(* PLC project Adressering.ecp, WAGO e!COCKPIT e!COCKPIT *)
(* stored: creationDateTime 2021-01-18T14:20:23.2110188, modificationDateTime 2021-01-18T11:51:27.6823754 *)

TYPE typVAV : STRUCT
  xReady : BOOL;  (* Status adr. *)
  xEnable : BOOL;  (* Enable MP blokk *)
  xAddress : BOOL;  (* Adresserer VAV *)
  xFailed : BOOL;  (* Tilbakemelding adressering (True = SerieNr inn og ut ikke stemmer) *)
  sSetStatus : STRING;  (* Status tilbakemelding naar adresseringen er i SET step *)
  sGetStatus : STRING;  (* Status tilbakemelding naar adresseringen er i GET step *)
  iSerialNr : typSerialNo;  (* Serie NR *)
  bPort : BYTE;  (* VAV Port *)
  bAddress : BYTE;  (* VAV Address *)
  rAirVolume_SP : REAL;  (* Settpunkt 0-100% *)
  rOutPosition : REAL;  (* Vinkel *)
  rOutAirVolume_perc : REAL;  (* Luftmengde i prosent *)
  rOutAirVolume_m3h : REAL;  (* Luftmengde i m3h *)
  wSensorValue : WORD;
  rVmin : REAL;
  rVmax : REAL;  (* Max vinkel *)
  xControlRangeIncreased : BOOL;
  xMecanicalOverload : BOOL;
  xActuatorHunting : BOOL;
  xSensorError : BOOL;
  xManualOpen : BOOL;
  xManualClose : BOOL;
  vMin : REAL;  (* Min luftmengde SP / 0-100 *)
  vNorm : REAL;  (* Settpunkt ved bevegelse / 0-100 *)
  vMax : REAL;  (* Maks luftmengde SP / 0-100 *)
  vSize : REAL;  (* Max kubikk *)
  vSetpoint_m3h : REAL;  (* SP% *)
  xdontoptimize : BOOL;  (* Fjerner VAV fra Optimizer *)
END_STRUCT;
END_TYPE

{attribute 'qualified_only'}
VAR_GLOBAL  (* STLV80_360 *)
  STLV80_A_360_6D201_SQ401 : typVAV := (xEnable := TRUE, vMin := 700, vNorm := 1400, vMax := 1400, vSize := 1750, bPort := 1, bAddress := 1, iSerialNr := (wYearAndWeek := 02045, wDayAndNumber := 50010, bTypeID := 158, bTestStation := 140));  (* / *)
  STLV80_A_360_6D301_SQ501 : typVAV := (xEnable := TRUE, vMin := 3200, vNorm := 3200, vMax := 3200, vSize := 5655, bPort := 1, bAddress := 2, iSerialNr := (wYearAndWeek := 02040, wDayAndNumber := 40202, bTypeID := 158, bTestStation := 153));  (* / *)
  STLV80_A_360_6A201_SQ401 : typVAV := (xEnable := TRUE, vMin := 2025, vNorm := 4050, vMax := 4050, vSize := 5655, bPort := 1, bAddress := 3, iSerialNr := (wYearAndWeek := 02040, wDayAndNumber := 40197, bTypeID := 158, bTestStation := 140));  (* / *)
  STLV80_A_360_6A201_SQ501 : typVAV := (xEnable := TRUE, vMin := 2700, vNorm := 2700, vMax := 2700, vSize := 5655, bPort := 1, bAddress := 4, iSerialNr := (wYearAndWeek := 02040, wDayAndNumber := 40201, bTypeID := 158, bTestStation := 159));  (* / *)
  STLV80_A_360_6C206_SQ501 : typVAV := (xEnable := TRUE, vMin := 300, vNorm := 300, vMax := 300, vSize := 700, bPort := 1, bAddress := 5, iSerialNr := (wYearAndWeek := 02105, wDayAndNumber := 10009, bTypeID := 158, bTestStation := 142));  (* / *)
  STLV80_A_360_6C206_SQ401 : typVAV := (xEnable := TRUE, vMin := 375, vNorm := 750, vMax := 750, vSize := 1750, bPort := 1, bAddress := 6, iSerialNr := (wYearAndWeek := 02045, wDayAndNumber := 50010, bTypeID := 158, bTestStation := 153));  (* / *)
  STLV80_A_360_7C201_SQ401 : typVAV := (xEnable := TRUE, vMin := 200, vNorm := 200, vMax := 200, vSize := 434, bPort := 1, bAddress := 7, iSerialNr := (wYearAndWeek := 02032, wDayAndNumber := 40145, bTypeID := 158, bTestStation := 158));  (* / *)
  STLV80_A_360_7C201_SQ501 : typVAV := (xEnable := TRUE, vMin := 400, vNorm := 400, vMax := 400, vSize := 700, bPort := 1, bAddress := 8, iSerialNr := (wYearAndWeek := 02042, wDayAndNumber := 10210, bTypeID := 158, bTestStation := 153));  (* / *)
  STLV80_A_360_6G201_SQ401 : typVAV := (xEnable := TRUE, vMin := 700, vNorm := 1400, vMax := 1400, vSize := 3619, bPort := 2, bAddress := 1, iSerialNr := (wYearAndWeek := 02042, wDayAndNumber := 10209, bTypeID := 158, bTestStation := 153));  (* / *)
  STLV80_A_360_6M201_SQ503 : typVAV := (xEnable := TRUE, vMin := 850, vNorm := 850, vMax := 850, vSize := 1060, bPort := 2, bAddress := 2, iSerialNr := (wYearAndWeek := 02005, wDayAndNumber := 20125, bTypeID := 158, bTestStation := 140));  (* / *)
  STLV80_A_360_6M201_SQ403 : typVAV := (xEnable := TRUE, vMin := 1225, vNorm := 2450, vMax := 2450, vSize := 5344, bPort := 2, bAddress := 3, iSerialNr := (wYearAndWeek := 02045, wDayAndNumber := 20003, bTypeID := 158, bTestStation := 140));  (* / *)
  STLV80_A_360_6M201_SQ402 : typVAV := (xEnable := TRUE, vMin := 700, vNorm := 1400, vMax := 1400, vSize := 4524, bPort := 2, bAddress := 4, iSerialNr := (wYearAndWeek := 02042, wDayAndNumber := 10207, bTypeID := 158, bTestStation := 153));  (* / *)
  STLV80_A_360_6M201_SQ502 : typVAV := (xEnable := TRUE, vMin := 3850, vNorm := 3850, vMax := 3850, vSize := 5655, bPort := 2, bAddress := 5, iSerialNr := (wYearAndWeek := 02040, wDayAndNumber := 40196, bTypeID := 158, bTestStation := 140));  (* / *)
  STLV80_A_360_6M201_SQ501 : typVAV := (xEnable := TRUE, vMin := 2600, vNorm := 2600, vMax := 2600, vSize := 5655, bPort := 2, bAddress := 6, iSerialNr := (wYearAndWeek := 02044, wDayAndNumber := 00121, bTypeID := 158, bTestStation := 164));  (* / *)
  STLV80_A_360_6M201_SQ401 : typVAV := (xEnable := TRUE, vMin := 900, vNorm := 1800, vMax := 1800, vSize := 5344, bPort := 2, bAddress := 7, iSerialNr := (wYearAndWeek := 02045, wDayAndNumber := 20006, bTypeID := 158, bTestStation := 140));  (* / *)
  STLV80_A_360_7O201_SQ401 : typVAV := (xEnable := TRUE, vMin := 200, vNorm := 200, vMax := 200, vSize := 700, bPort := 3, bAddress := 1, iSerialNr := (wYearAndWeek := 02032, wDayAndNumber := 40155, bTypeID := 158, bTestStation := 129));  (* / *)
  STLV80_A_360_7O201_SQ501 : typVAV := (xEnable := TRUE, vMin := 400, vNorm := 400, vMax := 400, vSize := 700, bPort := 3, bAddress := 2, iSerialNr := (wYearAndWeek := 02049, wDayAndNumber := 40093, bTypeID := 158, bTestStation := 142));  (* / *)
END_VAR

FUNCTION_BLOCK fbAutAd
  VAR_INPUT
    iSerialNr : typSerialNo;
    bPort : BYTE;
    bAddress : BYTE;
    xReset : BOOL;
    xNext : BOOL;
  END_VAR
  VAR_OUTPUT
    i : INT := 0;
    xFailed : BOOL;
    sSetStatus : STRING;
    sGetStatus : STRING;
  END_VAR
  VAR
    xLearn : BOOL;
    xRetry : BOOL;
    VAV_Addressing : fbMpBusAddressing;
  END_VAR

	//Resetter forgje VAVs verdier
	IF xReset THEN
		i:= 0;
		xRetry:= FALSE;
		xFailed:= FALSE;
		sSetStatus:= '';
		sGetStatus:= '';

//Begynner paa neste VAV
	ELSIF i<1 AND xNext THEN
		VAV_Addressing
		(
			bPortMpBus:= bPort,
			bAddress:= bAddress,
			typINSerialNo:= iSerialNr,
			xLearn:= xLearn
		);
		i:= 1;

//Skriver rett port og adresse til VAV naar blokken er klar
	ELSIF VAV_Addressing.xReady AND i=1 THEN
		VAV_Addressing
		(
			xSet:= TRUE,
			xLearn:= xLearn
		);
		i:= 2;

//Spoer etter serie nr som hoerer til port og adresse
	ELSIF VAV_Addressing.xReady AND i=2 THEN
		sSetStatus:= VAV_Addressing.sStatus;
		VAV_Addressing
		(
			xGetSerialNO:= TRUE,
			xLearn:= xLearn
		);
		i:= 3;

//Sjekker om serie nr. som tilhoerer port og adressen stemmer
	ELSIF VAV_Addressing.xReady AND i=3 THEN
		sGetStatus:= VAV_Addressing.sStatus;
		//Sjekker om serie nr stemmer
		IF xRetry AND VAV_Addressing.typOUTSerialNo.wYearAndWeek <> iSerialNr.wYearAndWeek OR VAV_Addressing.typOUTSerialNo.wDayAndNumber <> iSerialNr.wDayAndNumber OR VAV_Addressing.typOUTSerialNo.bTypeID <> iSerialNr.bTypeID OR VAV_Addressing.typOUTSerialNo.bTestStation <> iSerialNr.bTestStation THEN
			xRetry:= FALSE;
			xFailed:= TRUE;
			i:=4;
		ELSIF VAV_Addressing.typOUTSerialNo.wYearAndWeek <> iSerialNr.wYearAndWeek OR VAV_Addressing.typOUTSerialNo.wDayAndNumber <> iSerialNr.wDayAndNumber OR VAV_Addressing.typOUTSerialNo.bTypeID <> iSerialNr.bTypeID OR VAV_Addressing.typOUTSerialNo.bTestStation <> iSerialNr.bTestStation THEN
			xRetry:= TRUE;
			i:=1;
		ELSE
			i:=4;
		END_IF

//Resetter xSet og xGet, og Setter Port, adresse og serie nr. og henter status
	ELSE
		VAV_Addressing
		(
			bPortMpBus:= bPort,
			bAddress:= bAddress,
			typINSerialNo:= iSerialNr,
			xLearn:= xLearn,
			xSet:= FALSE,
			xGetSerialNO:= FALSE,
			xLearn:= xLearn
		);
	END_IF
				
END_FUNCTION_BLOCK

PROGRAM PRG_VAV_Adressering
  VAR
    xReset : BOOL;
    xRun : BOOL;
    xInit : BOOL := TRUE;
    Auto : fbAutAd;
    iLinje : INT;  (* Linje som skal adresseres *)
    iVAV : INT := 1;  (* VAV(adr.) som adresseres *)
  END_VAR

					IF xReset THEN
	Auto(xReset:= TRUE);
	xInit:= TRUE;
	xReset:= FALSE;
ELSIF xRun THEN

	IF STLV80_360.STLV80_A_360_6D201_SQ401.xAddress OR (iLinje = 1 AND iVAV = 1) THEN

		IF xInit THEN
			STLV80_360.STLV80_A_360_6D201_SQ401.xEnable:= FALSE;
			Auto(
				bPort:= STLV80_360.STLV80_A_360_6D201_SQ401.bPort,
				bAddress:= STLV80_360.STLV80_A_360_6D201_SQ401.bAddress,
				iSerialNr:= STLV80_360.STLV80_A_360_6D201_SQ401.iSerialNr,
				xNext:= TRUE,
				xReset:= FALSE
				);
			xInit:= FALSE;

		ELSIF Auto.i=4 THEN
			STLV80_360.STLV80_A_360_6D201_SQ401.sSetStatus:= Auto.sSetStatus;
				STLV80_360.STLV80_A_360_6D201_SQ401.sGetStatus:= Auto.sGetStatus;
				STLV80_360.STLV80_A_360_6D201_SQ401.xFailed:= Auto.xFailed;
				STLV80_360.STLV80_A_360_6D201_SQ401.xAddress:= FALSE;
				STLV80_360.STLV80_A_360_6D201_SQ401.xEnable:= TRUE;
				xReset:= TRUE;
				iVAV:=iVAV+1;

			ELSE
				Auto(xNext:= FALSE);
			END_IF

	ELSIF STLV80_360.STLV80_A_360_6D301_SQ501.xAddress OR (iLinje = 1 AND iVAV = 2) THEN

		IF xInit THEN
			STLV80_360.STLV80_A_360_6D301_SQ501.xEnable:= FALSE;
			Auto(
				bPort:= STLV80_360.STLV80_A_360_6D301_SQ501.bPort,
				bAddress:= STLV80_360.STLV80_A_360_6D301_SQ501.bAddress,
				iSerialNr:= STLV80_360.STLV80_A_360_6D301_SQ501.iSerialNr,
				xNext:= TRUE,
				xReset:= FALSE
				);
			xInit:= FALSE;

		ELSIF Auto.i=4 THEN
			STLV80_360.STLV80_A_360_6D301_SQ501.sSetStatus:= Auto.sSetStatus;
				STLV80_360.STLV80_A_360_6D301_SQ501.sGetStatus:= Auto.sGetStatus;
				STLV80_360.STLV80_A_360_6D301_SQ501.xFailed:= Auto.xFailed;
				STLV80_360.STLV80_A_360_6D301_SQ501.xAddress:= FALSE;
				STLV80_360.STLV80_A_360_6D301_SQ501.xEnable:= TRUE;
				xReset:= TRUE;
				iVAV:=iVAV+1;

			ELSE
				Auto(xNext:= FALSE);
			END_IF

	ELSIF STLV80_360.STLV80_A_360_6A201_SQ401.xAddress OR (iLinje = 1 AND iVAV = 3) THEN

		IF xInit THEN
			STLV80_360.STLV80_A_360_6A201_SQ401.xEnable:= FALSE;
			Auto(
				bPort:= STLV80_360.STLV80_A_360_6A201_SQ401.bPort,
				bAddress:= STLV80_360.STLV80_A_360_6A201_SQ401.bAddress,
				iSerialNr:= STLV80_360.STLV80_A_360_6A201_SQ401.iSerialNr,
				xNext:= TRUE,
				xReset:= FALSE
				);
			xInit:= FALSE;

		ELSIF Auto.i=4 THEN
			STLV80_360.STLV80_A_360_6A201_SQ401.sSetStatus:= Auto.sSetStatus;
				STLV80_360.STLV80_A_360_6A201_SQ401.sGetStatus:= Auto.sGetStatus;
				STLV80_360.STLV80_A_360_6A201_SQ401.xFailed:= Auto.xFailed;
				STLV80_360.STLV80_A_360_6A201_SQ401.xAddress:= FALSE;
				STLV80_360.STLV80_A_360_6A201_SQ401.xEnable:= TRUE;
				xReset:= TRUE;
				iVAV:=iVAV+1;

			ELSE
				Auto(xNext:= FALSE);
			END_IF

	ELSIF STLV80_360.STLV80_A_360_6A201_SQ501.xAddress OR (iLinje = 1 AND iVAV = 4) THEN

		IF xInit THEN
			STLV80_360.STLV80_A_360_6A201_SQ501.xEnable:= FALSE;
			Auto(
				bPort:= STLV80_360.STLV80_A_360_6A201_SQ501.bPort,
				bAddress:= STLV80_360.STLV80_A_360_6A201_SQ501.bAddress,
				iSerialNr:= STLV80_360.STLV80_A_360_6A201_SQ501.iSerialNr,
				xNext:= TRUE,
				xReset:= FALSE
				);
			xInit:= FALSE;

		ELSIF Auto.i=4 THEN
			STLV80_360.STLV80_A_360_6A201_SQ501.sSetStatus:= Auto.sSetStatus;
				STLV80_360.STLV80_A_360_6A201_SQ501.sGetStatus:= Auto.sGetStatus;
				STLV80_360.STLV80_A_360_6A201_SQ501.xFailed:= Auto.xFailed;
				STLV80_360.STLV80_A_360_6A201_SQ501.xAddress:= FALSE;
				STLV80_360.STLV80_A_360_6A201_SQ501.xEnable:= TRUE;
				xReset:= TRUE;
				iVAV:=iVAV+1;

			ELSE
				Auto(xNext:= FALSE);
			END_IF

	ELSIF STLV80_360.STLV80_A_360_6C206_SQ501.xAddress OR (iLinje = 1 AND iVAV = 5) THEN

		IF xInit THEN
			STLV80_360.STLV80_A_360_6C206_SQ501.xEnable:= FALSE;
			Auto(
				bPort:= STLV80_360.STLV80_A_360_6C206_SQ501.bPort,
				bAddress:= STLV80_360.STLV80_A_360_6C206_SQ501.bAddress,
				iSerialNr:= STLV80_360.STLV80_A_360_6C206_SQ501.iSerialNr,
				xNext:= TRUE,
				xReset:= FALSE
				);
			xInit:= FALSE;

		ELSIF Auto.i=4 THEN
			STLV80_360.STLV80_A_360_6C206_SQ501.sSetStatus:= Auto.sSetStatus;
				STLV80_360.STLV80_A_360_6C206_SQ501.sGetStatus:= Auto.sGetStatus;
				STLV80_360.STLV80_A_360_6C206_SQ501.xFailed:= Auto.xFailed;
				STLV80_360.STLV80_A_360_6C206_SQ501.xAddress:= FALSE;
				STLV80_360.STLV80_A_360_6C206_SQ501.xEnable:= TRUE;
				xReset:= TRUE;
				iVAV:=iVAV+1;

			ELSE
				Auto(xNext:= FALSE);
			END_IF

	ELSIF STLV80_360.STLV80_A_360_6C206_SQ401.xAddress OR (iLinje = 1 AND iVAV = 6) THEN

		IF xInit THEN
			STLV80_360.STLV80_A_360_6C206_SQ401.xEnable:= FALSE;
			Auto(
				bPort:= STLV80_360.STLV80_A_360_6C206_SQ401.bPort,
				bAddress:= STLV80_360.STLV80_A_360_6C206_SQ401.bAddress,
				iSerialNr:= STLV80_360.STLV80_A_360_6C206_SQ401.iSerialNr,
				xNext:= TRUE,
				xReset:= FALSE
				);
			xInit:= FALSE;

		ELSIF Auto.i=4 THEN
			STLV80_360.STLV80_A_360_6C206_SQ401.sSetStatus:= Auto.sSetStatus;
				STLV80_360.STLV80_A_360_6C206_SQ401.sGetStatus:= Auto.sGetStatus;
				STLV80_360.STLV80_A_360_6C206_SQ401.xFailed:= Auto.xFailed;
				STLV80_360.STLV80_A_360_6C206_SQ401.xAddress:= FALSE;
				STLV80_360.STLV80_A_360_6C206_SQ401.xEnable:= TRUE;
				xReset:= TRUE;
				iVAV:=iVAV+1;

			ELSE
				Auto(xNext:= FALSE);
			END_IF

	ELSIF STLV80_360.STLV80_A_360_7C201_SQ401.xAddress OR (iLinje = 1 AND iVAV = 7) THEN

		IF xInit THEN
			STLV80_360.STLV80_A_360_7C201_SQ401.xEnable:= FALSE;
			Auto(
				bPort:= STLV80_360.STLV80_A_360_7C201_SQ401.bPort,
				bAddress:= STLV80_360.STLV80_A_360_7C201_SQ401.bAddress,
				iSerialNr:= STLV80_360.STLV80_A_360_7C201_SQ401.iSerialNr,
				xNext:= TRUE,
				xReset:= FALSE
				);
			xInit:= FALSE;

		ELSIF Auto.i=4 THEN
			STLV80_360.STLV80_A_360_7C201_SQ401.sSetStatus:= Auto.sSetStatus;
				STLV80_360.STLV80_A_360_7C201_SQ401.sGetStatus:= Auto.sGetStatus;
				STLV80_360.STLV80_A_360_7C201_SQ401.xFailed:= Auto.xFailed;
				STLV80_360.STLV80_A_360_7C201_SQ401.xAddress:= FALSE;
				STLV80_360.STLV80_A_360_7C201_SQ401.xEnable:= TRUE;
				xReset:= TRUE;
				iVAV:=iVAV+1;

			ELSE
				Auto(xNext:= FALSE);
			END_IF

	ELSIF STLV80_360.STLV80_A_360_7C201_SQ501.xAddress OR (iLinje = 1 AND iVAV = 8) THEN

		IF xInit THEN
			STLV80_360.STLV80_A_360_7C201_SQ501.xEnable:= FALSE;
			Auto(
				bPort:= STLV80_360.STLV80_A_360_7C201_SQ501.bPort,
				bAddress:= STLV80_360.STLV80_A_360_7C201_SQ501.bAddress,
				iSerialNr:= STLV80_360.STLV80_A_360_7C201_SQ501.iSerialNr,
				xNext:= TRUE,
				xReset:= FALSE
				);
			xInit:= FALSE;

		ELSIF Auto.i=4 THEN
			STLV80_360.STLV80_A_360_7C201_SQ501.sSetStatus:= Auto.sSetStatus;
				STLV80_360.STLV80_A_360_7C201_SQ501.sGetStatus:= Auto.sGetStatus;
				STLV80_360.STLV80_A_360_7C201_SQ501.xFailed:= Auto.xFailed;
				STLV80_360.STLV80_A_360_7C201_SQ501.xAddress:= FALSE;
				STLV80_360.STLV80_A_360_7C201_SQ501.xEnable:= TRUE;
				xReset:= TRUE;
				iVAV:=iVAV+1;

			ELSE
				Auto(xNext:= FALSE);
			END_IF

	ELSIF STLV80_360.STLV80_A_360_6G201_SQ401.xAddress OR (iLinje = 2 AND iVAV = 1) THEN

		IF xInit THEN
			STLV80_360.STLV80_A_360_6G201_SQ401.xEnable:= FALSE;
			Auto(
				bPort:= STLV80_360.STLV80_A_360_6G201_SQ401.bPort,
				bAddress:= STLV80_360.STLV80_A_360_6G201_SQ401.bAddress,
				iSerialNr:= STLV80_360.STLV80_A_360_6G201_SQ401.iSerialNr,
				xNext:= TRUE,
				xReset:= FALSE
				);
			xInit:= FALSE;

		ELSIF Auto.i=4 THEN
			STLV80_360.STLV80_A_360_6G201_SQ401.sSetStatus:= Auto.sSetStatus;
				STLV80_360.STLV80_A_360_6G201_SQ401.sGetStatus:= Auto.sGetStatus;
				STLV80_360.STLV80_A_360_6G201_SQ401.xFailed:= Auto.xFailed;
				STLV80_360.STLV80_A_360_6G201_SQ401.xAddress:= FALSE;
				STLV80_360.STLV80_A_360_6G201_SQ401.xEnable:= TRUE;
				xReset:= TRUE;
				iVAV:=iVAV+1;

			ELSE
				Auto(xNext:= FALSE);
			END_IF

	ELSIF STLV80_360.STLV80_A_360_6M201_SQ503.xAddress OR (iLinje = 2 AND iVAV = 2) THEN

		IF xInit THEN
			STLV80_360.STLV80_A_360_6M201_SQ503.xEnable:= FALSE;
			Auto(
				bPort:= STLV80_360.STLV80_A_360_6M201_SQ503.bPort,
				bAddress:= STLV80_360.STLV80_A_360_6M201_SQ503.bAddress,
				iSerialNr:= STLV80_360.STLV80_A_360_6M201_SQ503.iSerialNr,
				xNext:= TRUE,
				xReset:= FALSE
				);
			xInit:= FALSE;

		ELSIF Auto.i=4 THEN
			STLV80_360.STLV80_A_360_6M201_SQ503.sSetStatus:= Auto.sSetStatus;
				STLV80_360.STLV80_A_360_6M201_SQ503.sGetStatus:= Auto.sGetStatus;
				STLV80_360.STLV80_A_360_6M201_SQ503.xFailed:= Auto.xFailed;
				STLV80_360.STLV80_A_360_6M201_SQ503.xAddress:= FALSE;
				STLV80_360.STLV80_A_360_6M201_SQ503.xEnable:= TRUE;
				xReset:= TRUE;
				iVAV:=iVAV+1;

			ELSE
				Auto(xNext:= FALSE);
			END_IF

	ELSIF STLV80_360.STLV80_A_360_6M201_SQ403.xAddress OR (iLinje = 2 AND iVAV = 3) THEN

		IF xInit THEN
			STLV80_360.STLV80_A_360_6M201_SQ403.xEnable:= FALSE;
			Auto(
				bPort:= STLV80_360.STLV80_A_360_6M201_SQ403.bPort,
				bAddress:= STLV80_360.STLV80_A_360_6M201_SQ403.bAddress,
				iSerialNr:= STLV80_360.STLV80_A_360_6M201_SQ403.iSerialNr,
				xNext:= TRUE,
				xReset:= FALSE
				);
			xInit:= FALSE;

		ELSIF Auto.i=4 THEN
			STLV80_360.STLV80_A_360_6M201_SQ403.sSetStatus:= Auto.sSetStatus;
				STLV80_360.STLV80_A_360_6M201_SQ403.sGetStatus:= Auto.sGetStatus;
				STLV80_360.STLV80_A_360_6M201_SQ403.xFailed:= Auto.xFailed;
				STLV80_360.STLV80_A_360_6M201_SQ403.xAddress:= FALSE;
				STLV80_360.STLV80_A_360_6M201_SQ403.xEnable:= TRUE;
				xReset:= TRUE;
				iVAV:=iVAV+1;

			ELSE
				Auto(xNext:= FALSE);
			END_IF

	ELSIF STLV80_360.STLV80_A_360_6M201_SQ402.xAddress OR (iLinje = 2 AND iVAV = 4) THEN

		IF xInit THEN
			STLV80_360.STLV80_A_360_6M201_SQ402.xEnable:= FALSE;
			Auto(
				bPort:= STLV80_360.STLV80_A_360_6M201_SQ402.bPort,
				bAddress:= STLV80_360.STLV80_A_360_6M201_SQ402.bAddress,
				iSerialNr:= STLV80_360.STLV80_A_360_6M201_SQ402.iSerialNr,
				xNext:= TRUE,
				xReset:= FALSE
				);
			xInit:= FALSE;

		ELSIF Auto.i=4 THEN
			STLV80_360.STLV80_A_360_6M201_SQ402.sSetStatus:= Auto.sSetStatus;
				STLV80_360.STLV80_A_360_6M201_SQ402.sGetStatus:= Auto.sGetStatus;
				STLV80_360.STLV80_A_360_6M201_SQ402.xFailed:= Auto.xFailed;
				STLV80_360.STLV80_A_360_6M201_SQ402.xAddress:= FALSE;
				STLV80_360.STLV80_A_360_6M201_SQ402.xEnable:= TRUE;
				xReset:= TRUE;
				iVAV:=iVAV+1;

			ELSE
				Auto(xNext:= FALSE);
			END_IF

	ELSIF STLV80_360.STLV80_A_360_6M201_SQ502.xAddress OR (iLinje = 2 AND iVAV = 5) THEN

		IF xInit THEN
			STLV80_360.STLV80_A_360_6M201_SQ502.xEnable:= FALSE;
			Auto(
				bPort:= STLV80_360.STLV80_A_360_6M201_SQ502.bPort,
				bAddress:= STLV80_360.STLV80_A_360_6M201_SQ502.bAddress,
				iSerialNr:= STLV80_360.STLV80_A_360_6M201_SQ502.iSerialNr,
				xNext:= TRUE,
				xReset:= FALSE
				);
			xInit:= FALSE;

		ELSIF Auto.i=4 THEN
			STLV80_360.STLV80_A_360_6M201_SQ502.sSetStatus:= Auto.sSetStatus;
				STLV80_360.STLV80_A_360_6M201_SQ502.sGetStatus:= Auto.sGetStatus;
				STLV80_360.STLV80_A_360_6M201_SQ502.xFailed:= Auto.xFailed;
				STLV80_360.STLV80_A_360_6M201_SQ502.xAddress:= FALSE;
				STLV80_360.STLV80_A_360_6M201_SQ502.xEnable:= TRUE;
				xReset:= TRUE;
				iVAV:=iVAV+1;

			ELSE
				Auto(xNext:= FALSE);
			END_IF

	ELSIF STLV80_360.STLV80_A_360_6M201_SQ501.xAddress OR (iLinje = 2 AND iVAV = 6) THEN

		IF xInit THEN
			STLV80_360.STLV80_A_360_6M201_SQ501.xEnable:= FALSE;
			Auto(
				bPort:= STLV80_360.STLV80_A_360_6M201_SQ501.bPort,
				bAddress:= STLV80_360.STLV80_A_360_6M201_SQ501.bAddress,
				iSerialNr:= STLV80_360.STLV80_A_360_6M201_SQ501.iSerialNr,
				xNext:= TRUE,
				xReset:= FALSE
				);
			xInit:= FALSE;

		ELSIF Auto.i=4 THEN
			STLV80_360.STLV80_A_360_6M201_SQ501.sSetStatus:= Auto.sSetStatus;
				STLV80_360.STLV80_A_360_6M201_SQ501.sGetStatus:= Auto.sGetStatus;
				STLV80_360.STLV80_A_360_6M201_SQ501.xFailed:= Auto.xFailed;
				STLV80_360.STLV80_A_360_6M201_SQ501.xAddress:= FALSE;
				STLV80_360.STLV80_A_360_6M201_SQ501.xEnable:= TRUE;
				xReset:= TRUE;
				iVAV:=iVAV+1;

			ELSE
				Auto(xNext:= FALSE);
			END_IF

	ELSIF STLV80_360.STLV80_A_360_6M201_SQ401.xAddress OR (iLinje = 2 AND iVAV = 7) THEN

		IF xInit THEN
			STLV80_360.STLV80_A_360_6M201_SQ401.xEnable:= FALSE;
			Auto(
				bPort:= STLV80_360.STLV80_A_360_6M201_SQ401.bPort,
				bAddress:= STLV80_360.STLV80_A_360_6M201_SQ401.bAddress,
				iSerialNr:= STLV80_360.STLV80_A_360_6M201_SQ401.iSerialNr,
				xNext:= TRUE,
				xReset:= FALSE
				);
			xInit:= FALSE;

		ELSIF Auto.i=4 THEN
			STLV80_360.STLV80_A_360_6M201_SQ401.sSetStatus:= Auto.sSetStatus;
				STLV80_360.STLV80_A_360_6M201_SQ401.sGetStatus:= Auto.sGetStatus;
				STLV80_360.STLV80_A_360_6M201_SQ401.xFailed:= Auto.xFailed;
				STLV80_360.STLV80_A_360_6M201_SQ401.xAddress:= FALSE;
				STLV80_360.STLV80_A_360_6M201_SQ401.xEnable:= TRUE;
				xReset:= TRUE;
				iVAV:=iVAV+1;

			ELSE
				Auto(xNext:= FALSE);
			END_IF

	ELSIF STLV80_360.STLV80_A_360_7O201_SQ401.xAddress OR (iLinje = 3 AND iVAV = 1) THEN

		IF xInit THEN
			STLV80_360.STLV80_A_360_7O201_SQ401.xEnable:= FALSE;
			Auto(
				bPort:= STLV80_360.STLV80_A_360_7O201_SQ401.bPort,
				bAddress:= STLV80_360.STLV80_A_360_7O201_SQ401.bAddress,
				iSerialNr:= STLV80_360.STLV80_A_360_7O201_SQ401.iSerialNr,
				xNext:= TRUE,
				xReset:= FALSE
				);
			xInit:= FALSE;

		ELSIF Auto.i=4 THEN
			STLV80_360.STLV80_A_360_7O201_SQ401.sSetStatus:= Auto.sSetStatus;
				STLV80_360.STLV80_A_360_7O201_SQ401.sGetStatus:= Auto.sGetStatus;
				STLV80_360.STLV80_A_360_7O201_SQ401.xFailed:= Auto.xFailed;
				STLV80_360.STLV80_A_360_7O201_SQ401.xAddress:= FALSE;
				STLV80_360.STLV80_A_360_7O201_SQ401.xEnable:= TRUE;
				xReset:= TRUE;
				iVAV:=iVAV+1;

			ELSE
				Auto(xNext:= FALSE);
			END_IF

	ELSIF STLV80_360.STLV80_A_360_7O201_SQ501.xAddress OR (iLinje = 3 AND iVAV = 2) THEN

		IF xInit THEN
			STLV80_360.STLV80_A_360_7O201_SQ501.xEnable:= FALSE;
			Auto(
				bPort:= STLV80_360.STLV80_A_360_7O201_SQ501.bPort,
				bAddress:= STLV80_360.STLV80_A_360_7O201_SQ501.bAddress,
				iSerialNr:= STLV80_360.STLV80_A_360_7O201_SQ501.iSerialNr,
				xNext:= TRUE,
				xReset:= FALSE
				);
			xInit:= FALSE;

		ELSIF Auto.i=4 THEN
			STLV80_360.STLV80_A_360_7O201_SQ501.sSetStatus:= Auto.sSetStatus;
				STLV80_360.STLV80_A_360_7O201_SQ501.sGetStatus:= Auto.sGetStatus;
				STLV80_360.STLV80_A_360_7O201_SQ501.xFailed:= Auto.xFailed;
				STLV80_360.STLV80_A_360_7O201_SQ501.xAddress:= FALSE;
				STLV80_360.STLV80_A_360_7O201_SQ501.xEnable:= TRUE;
				xReset:= TRUE;
				iVAV:=iVAV+1;

			ELSE
				Auto(xNext:= FALSE);
			END_IF

	ELSIF iVAV > 8 THEN
			iVAV:= 0;
		ELSIF iVAV > 0  THEN
			iVAV:= (iVAV+1);
		END_IF
END_IF

				
END_PROGRAM
